(* PLC project Senza_nome, Sconosciuto Senza_nome 1 *)
(* stored: creationDateTime 2026-08-24T10:02:07, modificationDateTime 2026-08-24T10:10:22 *)

PROGRAM program0
  VAR
    A AT %IX100.0 : BOOL;
    B AT %IX100.1 : BOOL;
    Q AT %QX100.0 : BOOL;
  END_VAR

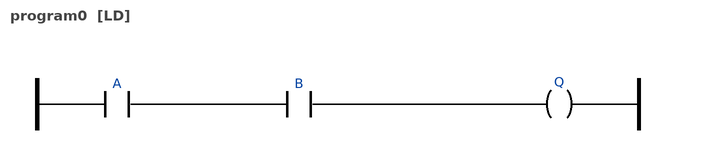
(* LD diagram, written out as Structured Text *)
Q := A AND B;
END_PROGRAM

CONFIGURATION Config0
  RESOURCE Res0 ON PLC
    TASK task0(INTERVAL := T#20ms, PRIORITY := 0);
    PROGRAM instance0 WITH task0 : program0;
  END_RESOURCE
END_CONFIGURATION
